FUNCTION F_LWORD_RTN : LWORD
VAR_INPUT
	stArg : ST_Arg;
END_VAR
VAR
	sysVar_Info : __SYSTEM.VAR_INFO;
END_VAR

sysVar_Info := __VARINFO(F_LWORD_RTN);
IF stArg.TypeClass = sysVar_Info.TypeClass THEN 
	F_LWORD_RTN := TO_LWORD(stArg.sValue);
	END_IF

END_FUNCTION

(* stored: Version 1.1.0.1, ProductVersion 3.1.4024.4
   POU F_LWORD_RTN: Id {20e52331-c065-44b9-a32d-5b8f1ab52d3e}, SpecialFunc None *)
